SUBAPPLICATION SwitchPic_5_3 (* Bild umschalten VT SK, AUX und VT Button; 5 Zustände *)
  (* Standard: 61499-2 *)
  (* Version 1.0, 2026-05-29, franz, Meisterschulen am Ostbahnhof *)
  PACKAGE MyLib::sys;
  IMPORT isobus::UT::Q::const::IDs::ID_NULL;
  IMPORT logiBUS::utils::sequence::schieber::SchieberStruct;
  IMPORT logiBUS::utils::sequence::schieber::const::iSTATES::Unknown;
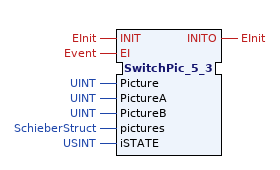
  EVENT_INPUT
    INIT : EInit; (* Initialization Request *)
    EI;
  END_EVENT
  EVENT_OUTPUT
    INITO : EInit; (* Initialization Confirm *)
  END_EVENT
  VAR_INPUT
    Picture : UINT; (* Object ID of the ObjectPointer to the Picture (SK) *)
    PictureA : UINT; (* Object ID of the ObjectPointer to the Picture (AUX) *)
    PictureB : UINT; (* Object ID of the ObjectPointer to the Picture (Button) *)
    pictures : logiBUS::utils::sequence::schieber::SchieberStruct := (Unknown := ID_NULL, Closed := ID_NULL, Opening := ID_NULL, Opened := ID_NULL, Closing := ID_NULL); (* the single Pictures *)
    iSTATE : USINT := Unknown;
  END_VAR
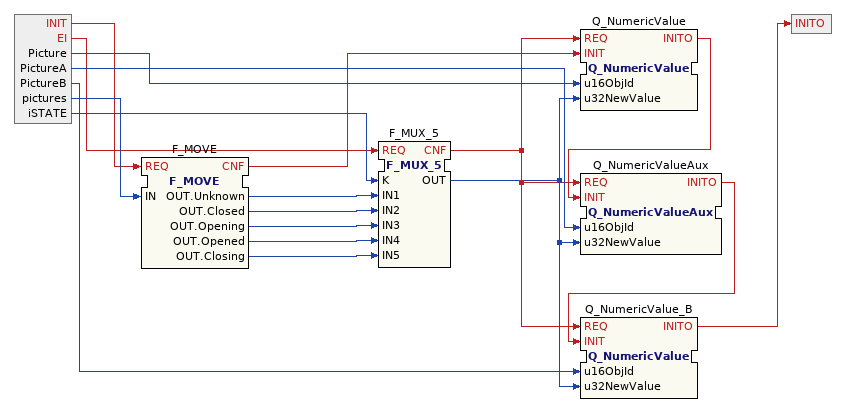
  FBS
    Q_NumericValue : isobus::UT::Q::Q_NumericValue;
    Q_NumericValueAux : isobus::UT::Q::Q_NumericValueAux;
    Q_NumericValue_B : isobus::UT::Q::Q_NumericValue;
    F_MOVE : iec61131::selection::F_MOVE; {SET_ATTRIBUTE(DataType, logiBUS::utils::sequence::schieber::SchieberStruct)}
    F_MUX_5 : iec61131::selection::F_MUX_5;
  END_FBS
  EVENT_CONNECTIONS
    EI TO F_MUX_5.REQ;
    F_MUX_5.CNF TO Q_NumericValue.REQ;
    F_MUX_5.CNF TO Q_NumericValueAux.REQ;
    F_MUX_5.CNF TO Q_NumericValue_B.REQ;
    INIT TO F_MOVE.REQ;
    F_MOVE.CNF TO Q_NumericValue.INIT;
    Q_NumericValue.INITO TO Q_NumericValueAux.INIT;
    Q_NumericValueAux.INITO TO Q_NumericValue_B.INIT;
    Q_NumericValue_B.INITO TO INITO;
  END_CONNECTIONS
  DATA_CONNECTIONS
    Picture TO Q_NumericValue.u16ObjId;
    PictureA TO Q_NumericValueAux.u16ObjId;
    PictureB TO Q_NumericValue_B.u16ObjId;
    pictures TO F_MOVE.IN;
    iSTATE TO F_MUX_5.K;
    F_MUX_5.OUT TO Q_NumericValue.u32NewValue;
    F_MUX_5.OUT TO Q_NumericValueAux.u32NewValue;
    F_MUX_5.OUT TO Q_NumericValue_B.u32NewValue;
    F_MOVE.OUT.Unknown TO F_MUX_5.IN1;
    F_MOVE.OUT.Closed TO F_MUX_5.IN2;
    F_MOVE.OUT.Opening TO F_MUX_5.IN3;
    F_MOVE.OUT.Opened TO F_MUX_5.IN4;
    F_MOVE.OUT.Closing TO F_MUX_5.IN5;
  END_CONNECTIONS
END_SUBAPPLICATION
